Fanuc KAREL source: kb00087.KL

-- PROVISIONAL review KL for V770-1; original PC SHA256 3825b7af5166ae4f271a6bee1fbf5169888bb834a5cace2432bb5c47810979f5
-- Incomplete behavior may be omitted. Consult companion uncertainty JSON. Do not deploy.
PROGRAM KB00087
%NOLOCKGROUP
BEGIN
  -- UNRESOLVED_PC offsets 5-12; opcodes 9D,23
  -- UNRESOLVED_PC offsets 17-24; opcodes 9D,23
  -- UNRESOLVED_PC offsets 29-59; opcodes 27,22,22,27,9D,31,7E,4A
  -- UNRESOLVED_PC offsets 64-68; opcodes 7F
END KB00087
